FUNCTION_BLOCK ABSTRACT FB_ActorContinous EXTENDS FB_Actor2Point
VAR_INPUT
	fSetPointAutomatic	: REAL; //unit depending setpoint
END_VAR
VAR_OUTPUT
END_VAR
VAR
	{attribute 'OPC.UA.DA' := '1'}
	setSetPoint : ST_SetSetPoint;
	{attribute 'OPC.UA.DA' := '1'}
	setPointState : ST_SetPointState;
	
	//internal variables
	fSetPoint	    : REAL; //actual set setpoint
	aSetPointLimits	: ARRAY[1..2] OF REAL; //control mode and unit depending setpoint limits that are set by abstract method SetSetPointLimits() in a subclass 
END_VAR

PROPERTY fOperatingPoint : REAL
GET
fOperatingPoint := setPointState.fOperatingPoint;
END_GET
END_PROPERTY

METHOD PROTECTED MAIN : BOOL // Method that calls all needed function block methods
VAR_INPUT
END_VAR
SelectControlMode();
SetSetPointLimits();
SetPointCheck();
END_METHOD

METHOD PROTECTED SelectControlMode : BOOL
VAR_INPUT
END_VAR
SUPER^.SelectControlMode();

//add changing set point to method
IF control.bManualModeActivated THEN
	fsetPoint := setSetPoint.fSetPointManual;
ELSIF control.bAlgorithmModeActivated AND bAlgorithmPermission THEN
	fsetPoint := setSetPoint.fSetPointAlgorithm;
ELSE
	fsetPoint := fSetPointAutomatic;
END_IF
END_METHOD

METHOD PRIVATE SetPointCheck : BOOL
VAR
END_VAR
fSetPoint := MAX(fSetPoint, aSetPointLimits[1]);
fSetPoint := MIN(fSetPoint, aSetPointLimits[2]);
END_METHOD

METHOD PROTECTED ABSTRACT SetSetPointLimits : BOOL
VAR_INPUT
END_VAR
//set control mode depending setpoint limits -> aSetPointLimits
END_METHOD

END_FUNCTION_BLOCK

(* stored: Version 1.1.0.1, ProductVersion 3.1.4024.9
   POU FB_ActorContinous: Id {c8bff7e9-c02c-4471-8259-14c86f2cd564}, SpecialFunc None
   Property fOperatingPoint: Id {9e55e02a-e000-449d-ace8-c0c0318e8e4a}
   Get Get: Id {646b79d7-340e-449c-a059-1923543a0f71}
   Method MAIN: Id {7c71e98c-e88b-49de-b162-405ba243d74c}
   Method SelectControlMode: Id {9487b088-9bc5-4a7e-8bf7-9767eafe3f05}
   Method SetPointCheck: Id {a788f595-bc97-42ed-a5e1-110d1f06de83}
   Method SetSetPointLimits: Id {156a380a-be13-4137-b0ba-36981904d328} *)
